FUNCTION_BLOCK FB_SlaveCtrlPrecisionTest EXTENDS FB_SlaveArmCtrlBase
VAR_INPUT
END_VAR
VAR_OUTPUT
END_VAR
VAR
	//arm id
	m_armId:INT;	
	
	//Precision calculation pre matrix
	m_frontPose:ST_Frame;
	
	//Precision calculation post matrix
	m_endPose:ST_Frame;
	
	//single arm pose
	m_slaveArmPose:ST_Frame;
	
	//control mode:  1---Joint space single point motion   2---Continuous joint space motion   3---Single point motion in operating space
	//4---Continuous motion in operating space   5---precision test   6---back to origin position
	m_controlMode:INT:=1;
	
	//test step
	m_testStep:INT;
	
	//DH joint position
	m_initDHPos,m_startDHPos,m_endDHPos :Vec6d;
	
	//startJntPos,endJntPos :Vec8d;
	m_initJntPos,m_startJntPos,m_endJntPos :Vec8d;
	
	//Trajectory planner
	m_Planner: FB_TrajMoveJ;
	
	//motion parameters
	m_maxjntVel,m_maxjntAcc,m_maxjntJerk:Vec8d;
	
	// joint velocity limit
	m_DHJntVel :ARRAY[1..6] OF LREAL :=[1, 1, 0.5, 1,1,1];
	m_maxDHJntVel :ARRAY[1..6] OF LREAL :=[1, 1, 0.5, 1,1,1];	
	m_velFactor:ARRAY[1..2] OF LREAL:=[0.1,1];//lowVel  highVel
	
	//time
	m_time:LREAL;
	
	//joint motion incresement
	m_DHjntInc:Vec6d;
	
	//moiton parameters
	m_jntMotionDir:Vec6i:=[0,0,0,0,0,0];
	m_jntVel:Vec6d:=[0.1,0.1,0.01,0.2,0.2,0.2];
	
	//motion start
	m_startMotion:BOOL;
	m_startMotionLast:BOOL;
	
	//target spatial position
	m_targetSpatialPos:ST_Frame;
	
	//spatial motion parameters
	m_spatialMotionDir:Vec6i;
	m_spatialVel:Vec6d;
	
	//spatial position incresement
	m_spatialPosInc:Vec6d;
	
	//initial spatial position
	m_initSpatialPos:ST_Frame;
	
	//target position variables
	m_posInc:Vec3d;
	m_axis:Vec3d;
	m_angle:LREAL;
	
	//accuracy test variables
	m_pointNum:INT;
	m_pointSum:INT;
	m_motionCycleNum:INT;
	m_targetPosArr:ARRAY[1..5] OF ST_Frame;
	
	//Has the inverse kinematics been successfully solved
	m_IKSucceed:BOOL;	
	
	//Numerical method for inverse solution of related variables
	//m_cmdCartPose:ST_Frame;
	m_slavePosErr :Vec3d;
	m_slaveRotErr :Mat3d;
	m_errAngle : LREAL;
	m_errAxisLocal, m_errAxis :Vec3d;
	m_masterSlavePoseError :Vec6d;
	
	// pose track control kp
	m_posTrackKp :REAL := 100;
	m_oriTrackKp :REAL := 100;
	
	// velocity for slave to track motion
	m_slaveCmdVel, m_slaveCmdWVel : Vec3d;
	invJaco :Mat6d;
	
	//spatial velocity limit
	m_linearVelLimit:LREAL:=0.1;
	m_angularVelLimit:LREAL:=5*g_deg2Rad;
	
	// simulated DH joint position
	m_simDHJntPos : Vec6d;
	
	// simulated slave twist of DH joint
	m_simDHJointVel :Vec6d;
	
	// command joint position filter
	m_cmdJntPosLpf:ARRAY[1..8] OF FB_LowPassFilter;
	
	// filter cut-off frequency for control
	m_macroCmdJntPosLpfCutoffFreq : LREAL :=5;
	m_microCmdJntPosLpfCutoffFreq : LREAL :=15;
	
	//position and posture error limit
	m_distErrLimit:LREAL:=0.001*0.1;
	m_poseErrLimit:LREAL:=0.01*g_deg2Rad;
	m_delayTimeLimit:LREAL:=1;
	m_errTime:LREAL;
	
	//original joint position
	m_originJntPos:Vec6d;
	
	//motion status
	m_motionFinished:BOOL;
END_VAR

METHOD accuracyTest : BOOL
VAR_INPUT
	// slave arm data
	i_slaveArm :FB_SlaveArm;
END_VAR

(*
CASE m_testStep OF
	0: //data initial		
		m_targetSpatialPos:=m_targetPosArr[m_pointNum];
		m_startDHPos:=i_slaveArm.curDHJntPos;
		m_IKSucceed:=i_slaveArm.inverseKinematic(i_targetSpatialPos:= m_targetSpatialPos, i_startDHJntPos:= m_startDHPos, o_outputDHJntPos=> m_endDHPos);
		IF (m_IKSucceed=FALSE) THEN
			m_testStep:=30;
		END_IF
		
		m_startJntPos:=i_slaveArm.curJntPos;	
		i_slaveArm.instrument.instruIK(m_endDHPos,0, o_jntPos=>m_endJntPos);
		m_Planner.init(i_startJntPos:= m_startJntPos, 	i_targetJntPos:= m_endJntPos, 	i_maxJntVel:= m_maxjntVel, 	i_maxJntAcc:= m_maxjntAcc, 	i_maxJntJerk:= m_maxjntJerk);
		IF (m_Planner.isGene=FALSE) THEN
			m_testStep:=30;
		ELSE
			m_time:=0; m_testStep:=10;
		END_IF		
		
		
	10: //start the motion
		m_time:=m_time+g_slaveArmCtrlCycleTime;
		m_Planner.evaluate(t:= m_time, jntPos=> m_cmdJntPos, jntVel=> m_cmdJntVel, jntAcc=> m_cmdJntAcc);
		IF (m_time>m_Planner.duration) THEN
			m_testStep:=20;			
		END_IF
		
		
	20: //Record the motion cycle
		m_pointNum:=m_pointNum+1;
		IF (m_pointNum>m_pointSum) THEN
			m_pointNum:=1;
			m_motionCycleNum:=m_motionCycleNum+1;
			IF (m_motionCycleNum>5) THEN
				m_testStep:=30;
			ELSE
				m_testStep:=0;
			END_IF
		ELSE
			m_testStep:=0;
		END_IF
		
	
	30: //stop
		m_testStep:=-1;		
END_CASE
*)
END_METHOD

METHOD accuracyTest_iter : BOOL
VAR_INPUT
	// slave arm data
	i_slaveArm :FB_SlaveArm;
END_VAR

CASE m_testStep OF
	0: //data initial		
		m_targetSpatialPos:=m_targetPosArr[m_pointNum];
		m_cmdCartPose:=m_targetSpatialPos;
		numericalIK(i_slaveArm);
		
		//Determine if the error is less than the set value
		IF (norm(m_slavePosErr)<m_distErrLimit) AND (m_errAngle<m_poseErrLimit) THEN
			m_errTime:=m_errTime+g_slaveArmCtrlCycleTime;
			IF (m_errTime>m_delayTimeLimit) THEN
				m_errTime:=0;
				m_testStep:=15;
			END_IF
		ELSE
			m_errTime:=0;
		END_IF
	
		
	15: //Waiting for confirmation and measurement
		IF (GVL_AccuracyTestVar.g_nextStep[m_armId]=TRUE) THEN
			GVL_AccuracyTestVar.g_nextStep[m_armId]:=FALSE;
			m_testStep:=20;
		END_IF
		
	
	20: //Record the motion cycle
		m_pointNum:=m_pointNum+1;
		IF (m_pointNum>m_pointSum) THEN
			m_pointNum:=1;
			m_motionCycleNum:=m_motionCycleNum+1;
			IF (m_motionCycleNum>GVL_AccuracyTest.g_testMotCycNum) THEN
				m_testStep:=30;
			ELSE
				m_testStep:=0;
			END_IF
		ELSE
			m_testStep:=0;
		END_IF
	
	
	30: //stop
		m_testStep:=-1;	
		m_motionFinished:=TRUE;	
END_CASE
END_METHOD

METHOD back2origin : BOOL
VAR_INPUT
	// slave arm data
	i_slaveArm :FB_SlaveArm;
END_VAR

CASE m_testStep OF
	0: //Trajectory parameter initialization
		m_startJntPos:=i_slaveArm.curJntPos;
		m_endDHPos:=m_originJntPos;		
		i_slaveArm.instrument.instruIK(m_endDHPos,0, o_jntPos=>m_endJntPos);
		m_Planner.init(i_startJntPos:= m_startJntPos, 	i_targetJntPos:= m_endJntPos, 	i_maxJntVel:= m_maxjntVel, 	i_maxJntAcc:= m_maxjntAcc, 	i_maxJntJerk:= m_maxjntJerk);
		IF (m_Planner.isGene=FALSE) THEN
			m_testStep:=20;
		ELSE
			m_time:=0; m_testStep:=10;
		END_IF		
		
		
	10: //start motion
		m_time:=m_time+g_slaveArmCtrlCycleTime;
		m_Planner.evaluate(t:= m_time, jntPos=> m_cmdJntPos, jntVel=> m_cmdJntVel, jntAcc=> m_cmdJntAcc);
		m_simJntPos:=m_cmdJntPos; //copy value to sim jntpos
		IF (m_time>m_Planner.duration) THEN
			m_testStep:=20;
		END_IF		
		
		
	20: //end the motion
		m_testStep:=-1;		
		m_motionFinished:=TRUE;
END_CASE
END_METHOD

// override this function in each exact controller
METHOD PROTECTED calcCmdJntPos : BOOL
VAR_IN_OUT CONSTANT
	// endoscope pose in cart coordinate
	i_endoscopePose : ST_Frame;
	
	// master arm data
	i_masterStatus :ST_MasterStatus;
	
	// setup arm data
	i_setupStatus: ST_SetupStatus;
	
	// slave arm data
	i_slaveArm :FB_SlaveArm;
END_VAR

VAR
	i:INT;
	tmpFrame:ST_Frame;
	r_angle:LREAL;
END_VAR

//Basic information update---front pose frame and end pose frame 
tmpFrame:=invFrame(i_endoscopePose);
i:=i_slaveArm.armIdx;
m_frontPose:=transform(tmpFrame,i_setupStatus.m_curEndPose[i]);
m_endPose.m_pos:=g_zeroVec3d;  m_endPose.m_rot:=g_eye3d;
m_slaveArmPose:=i_slaveArm.curCartPose;


//copy to global variables
GVL_AccuracyTestVar.g_frontPose[m_armId]:=m_frontPose;
GVL_AccuracyTestVar.g_endPose[m_armId]:=m_endPose;
GVL_AccuracyTestVar.g_slaveArmPose[m_armId]:=m_slaveArmPose;


//Initialization of motion parameters
m_startMotion:=GVL_AccuracyTestVar.g_startMotion[m_armId];
IF (m_startMotionLast=FALSE) AND (m_startMotion=TRUE) THEN
	motionParamInit(i_slaveArm);
END_IF
m_startMotionLast:=m_startMotion;


//Select different programs based on different control modes
IF (m_startMotion=TRUE) THEN
	IF (m_controlMode=1) THEN
		//jntSinglePoint(i_slaveArm);
		
	ELSIF (m_controlMode=2) THEN
		jntContinuousPoint(i_slaveArm);
		
	ELSIF (m_controlMode=3) THEN
		//spaceSinglePoint_iter(i_slaveArm);
		
	ELSIF (m_controlMode=4) THEN
		spaceContinuousPoint_iter(i_slaveArm);
		
	ELSIF (m_controlMode=5) THEN
		accuracyTest_iter(i_slaveArm);
		
	ELSIF (m_controlMode=6) THEN
		back2origin(i_slaveArm);
	END_IF
END_IF


//show the motion step
IF (m_controlMode=5) THEN
	GVL_AccuracyTestVar.g_curStep[m_armId]:=m_testStep;
	GVL_AccuracyTestVar.g_testPointId[m_armId]:=m_pointNum;
	GVL_AccuracyTestVar.g_testCycleId[m_armId]:=m_motionCycleNum;
ELSE
	GVL_AccuracyTestVar.g_curStep[m_armId]:=-1;
	GVL_AccuracyTestVar.g_testPointId[m_armId]:=0;
	GVL_AccuracyTestVar.g_testCycleId[m_armId]:=0;
END_IF



// feedback the motion status
IF (m_controlMode=1) OR (m_controlMode=3) OR (m_controlMode=5) OR (m_controlMode=6) THEN
	IF (m_testStep=-1) AND (m_motionFinished=TRUE) THEN
		m_controlMode:=0;
		GVL_AccuracyTestVar.g_controlMode[m_armId]:=0;	
	END_IF
ELSIF (m_controlMode=2) OR (m_controlMode=4) THEN
	IF (m_startMotion=FALSE) THEN
		m_controlMode:=0;
		GVL_AccuracyTestVar.g_controlMode[m_armId]:=0;
	END_IF
END_IF
END_METHOD

// override this function in each exact controller
// NOTICE: set joint control mode here, and do some initialization if needed
METHOD PUBLIC init : BOOL
VAR_IN_OUT CONSTANT
	i_slaveArm	:FB_SlaveArm;
END_VAR
VAR_IN_OUT 
	r_slaveArmCtrlCmd :ST_SlaveArmCtrlCmds;	
END_VAR

VAR
	
END_VAR
SUPER^.Init(i_slaveArm,r_slaveArmCtrlCmd);

//variable initialization
m_armId:=i_slaveArm.armIdx;

//motion parameters initial
motionParamInit(i_slaveArm);
END_METHOD

METHOD PROTECTED jntContinuousPoint : BOOL
VAR_INPUT
	// slave arm data
	i_slaveArm :FB_SlaveArm;
END_VAR

VAR
	i:INT;
END_VAR

//joint motion incresement calculation
FOR i:=1 TO 6 BY 1 DO
	m_DHjntInc[i]:=m_DHjntInc[i]+m_jntMotionDir[i]*m_jntVel[i]*g_slaveArmCtrlCycleTime;
END_FOR

//determine DH joint position
vecAdd(m_initDHPos,m_DHjntInc,m_endDHPos);
i_slaveArm.instrument.instruIK(m_endDHPos,0, o_jntPos=>m_endJntPos);

//copy the value
m_cmdJntPos:=m_endJntPos;
m_simJntPos:=m_cmdJntPos; //copy value to sim jntpos
END_METHOD

METHOD jntSinglePoint : BOOL
VAR_INPUT
	// slave arm data
	i_slaveArm :FB_SlaveArm;
END_VAR

CASE m_testStep OF
	0: //Trajectory parameter initialization
		m_startJntPos:=i_slaveArm.curJntPos;
		m_endDHPos:=GVL_AccuracyTestVar.g_targetJntPos[m_armId];
		
		i_slaveArm.instrument.instruIK(m_endDHPos,0, o_jntPos=>m_endJntPos);
		m_Planner.init(i_startJntPos:= m_startJntPos, 	i_targetJntPos:= m_endJntPos, 	i_maxJntVel:= m_maxjntVel, 	i_maxJntAcc:= m_maxjntAcc, 	i_maxJntJerk:= m_maxjntJerk);
		IF (m_Planner.isGene=FALSE) THEN
			m_testStep:=20;
		ELSE
			m_time:=0; m_testStep:=10;
		END_IF		
		
		
	10: //start motion
		m_time:=m_time+g_slaveArmCtrlCycleTime;
		m_Planner.evaluate(t:= m_time, jntPos=> m_cmdJntPos, jntVel=> m_cmdJntVel, jntAcc=> m_cmdJntAcc);
		m_simJntPos:=m_cmdJntPos; //copy value to sim jntpos
		IF (m_time>m_Planner.duration) THEN
			m_testStep:=20;
		END_IF		
		
		
	20: //end the motion
		m_testStep:=-1;		
		m_motionFinished:=TRUE;
END_CASE
END_METHOD

METHOD motionParamInit : BOOL
VAR_INPUT
	// slave arm data
	i_slaveArm :FB_SlaveArm;
END_VAR
VAR
	i,j:INT;
	poseVec:Vec6d;
	originPose:ST_Frame;
END_VAR
m_testStep:=0;
m_time:=0;
m_controlMode:=GVL_AccuracyTestVar.g_controlMode[m_armId];
m_motionFinished:=FALSE;


//update the joint velocity
IF (m_controlMode=3) OR (m_controlMode=5) THEN
	vecMultiNum(m_DHJntVel,m_velFactor[1],m_maxDHJntVel); //low velocity
ELSIF (m_controlMode=4) THEN	
	vecMultiNum(m_DHJntVel,m_velFactor[2],m_maxDHJntVel); //high velocity
ELSE
	m_maxDHJntVel:=m_DHJntVel; //original velocity
END_IF


//joint continuous motion parameters
m_initDHPos:=i_slaveArm.curDHJntPos;
m_DHjntInc:=g_zeroVec6d;
m_jntMotionDir:=GVL_AccuracyTestVar.g_jntMotionDir[m_armId];
m_jntVel:=GVL_AccuracyTestVar.g_jntVel[m_armId];
FOR i:=1 TO 6 BY 1 DO
	m_jntVel[i]:=LIMIT(-0.1,m_jntVel[i],0.1);
END_FOR
m_jntVel[3]:=LIMIT(-0.01,m_jntVel[3],0.01);


//spatial continuous motion parameters
m_spatialMotionDir:=GVL_AccuracyTestVar.g_spatialMotionDir[m_armId];
m_spatialVel:=GVL_AccuracyTestVar.g_spatialVel[m_armId];
m_initSpatialPos:=i_slaveArm.curCartPose;
m_spatialPosInc:=g_zeroVec6d;
FOR i:=1 TO 3 BY 1 DO
	m_spatialVel[i]:=LIMIT(-0.01,m_spatialVel[i],0.01);
END_FOR
FOR i:=4 TO 6 BY 1 DO
	m_spatialVel[i]:=LIMIT(-0.1,m_spatialVel[i],0.1);
END_FOR


//velocity---acceleration---jerk
vecMultiNum(GVL_SlaveMotorParameters.g_maxJntVel,0.2,m_maxjntVel);
vecMultiNum(m_maxjntVel,3,m_maxjntAcc);
vecMultiNum(m_maxjntAcc,3,m_maxjntJerk);


//accuracy test variables
m_pointNum:=1;
m_pointSum:=GVL_AccuracyTest.g_testPointNum;
m_motionCycleNum:=1;
m_errTime:=0;


//original joint position
m_originJntPos:=GVL_AccuracyTest.g_originJntPos;


//Obtain the position and posture of the test point location
FOR i:=1 TO 5 BY 1 DO
	FOR j:=1 TO 6 BY 1 DO
		poseVec[j]:=GVL_AccuracyTest.g_testSpacePoint[i,j];
	END_FOR
	xyzrpy2Frame(i_posVec:= poseVec, o_frame=> m_targetPosArr[i]);
	
	i_slaveArm.forwardKinematic(i_DHJntPos:= m_originJntPos, r_cartPose:= originPose);
	m_targetPosArr[i].m_rot:=originPose.m_rot;
END_FOR


// init filter
FOR i:=1 TO 3 DO
	m_cmdJntPosLpf[i].init(1, m_macroCmdJntPosLpfCutoffFreq, g_slaveArmCtrlFreq);
END_FOR
FOR i:=4 TO g_sJntNum DO
	m_cmdJntPosLpf[i].init(1, m_microCmdJntPosLpfCutoffFreq, g_slaveArmCtrlFreq);
END_FOR
END_METHOD

METHOD numericalIK : BOOL
VAR_INPUT
	// slave arm data
	i_slaveArm :FB_SlaveArm;
END_VAR

VAR
	i:INT;
	tmpMat3d:Mat3d;
	linearVelScale:LREAL;
	angularVelScale:LREAL;
END_VAR

		//Solve the error term
		vecSub(m_cmdCartPose.m_pos, i_slaveArm.simCartPose.m_pos, m_slavePosErr);
		matTranspose(i_slaveArm.simCartPose.m_rot, tmpMat3d);
		matMultiply(tmpMat3d, m_cmdCartPose.m_rot, m_slaveRotErr);
		rot2AngAxis(m_slaveRotErr, angle=>m_errAngle, axis=>m_errAxisLocal);
		matMultiVec(i_slaveArm.simCartPose.m_rot, m_errAxisLocal, m_errAxis);
		
		// pose track control
		vecMultiNum(m_slavePosErr, m_posTrackKp, m_slaveCmdVel);
		vecMultiNum(m_errAxis, m_errAngle*m_oriTrackKp, m_slaveCmdWVel);
		
		
		//Limit spatial linear velocity and angular velocity
		linearVelScale:=norm(m_slaveCmdVel)/m_linearVelLimit;
		angularVelScale:=norm(m_slaveCmdWVel)/m_angularVelLimit;	
		IF (linearVelScale)>1 THEN
			vecSelfMultiNum(m_slaveCmdVel,1.0/linearVelScale);
		END_IF
		IF (angularVelScale)>1 THEN
			vecSelfMultiNum(m_slaveCmdWVel,1.0/angularVelScale);
		END_IF
		
		
		// final command twist
		FOR i:=1 TO 3 DO 
			m_cmdCartTwist[i] := m_slaveCmdVel[i];
			m_cmdCartTwist[i+3] := m_slaveCmdWVel[i];
		END_FOR
		
		// compute command velocity for DH joints
		invJaco := i_slaveArm.simJacoInv;
		matMultiVec(invJaco, m_cmdCartTwist, m_simDHJointVel);
		
		// limit DH joints velocity and integrate command DH joint position
		FOR i:=1 TO 6 DO 
			m_simDHJointVel[i] := LIMIT(-m_maxDHJntVel[i], m_simDHJointVel[i], m_maxDHJntVel[i]);
			
			m_simDHJntPos[i] := i_slaveArm.simDHJntPos[i] + m_simDHJointVel[i]*g_slaveArmCtrlCycleTime;
			IF (m_simDHJntPos[i]>GVL_SlaveMotorParameters.g_maxDHJntPos[i]) OR (m_simDHJntPos[i]<GVL_SlaveMotorParameters.g_minDHJntPos[i]) THEN
				m_simDHJointVel[i]:=0;
				m_simDHJntPos[i] := i_slaveArm.simDHJntPos[i];
			END_IF
		END_FOR
		
		// calculate target motor joint position/velocity from DH joint position
		i_slaveArm.instrument.instruIK(m_simDHJntPos,0, o_jntPos=>m_simJntPos);
		
		// filt command joint position
		FOR i:=1 TO g_sJntNum DO 
			//m_cmdJntPos[i] := m_cmdJntPosLpf[i].run(m_simJntPos[i]);
		END_FOR
		m_cmdJntPos:=m_simJntPos;
END_METHOD

METHOD rpy2rot : BOOL
VAR_INPUT
	i_rpy:Vec3d;
END_VAR

VAR_OUTPUT
	o_rot:Mat3d;
END_VAR

VAR
	rot_x,rot_y,rot_z:LREAL;
	alpha,beta,gama:LREAL;
	matrix_out:ARRAY[1..3,1..3] OF LREAL;
END_VAR

alpha:=rot_z;
beta:=rot_y;
gama:=rot_x;

matrix_out[1,1]:=COS(alpha)*COS(beta);
matrix_out[2,1]:=SIN(alpha)*COS(beta);
matrix_out[3,1]:=-SIN(beta);

matrix_out[1,2]:=COS(alpha)*SIN(beta)*SIN(gama)-SIN(alpha)*COS(gama);
matrix_out[2,2]:=SIN(alpha)*SIN(beta)*SIN(gama)+COS(alpha)*COS(gama);
matrix_out[3,2]:=COS(beta)*SIN(gama);

matrix_out[1,3]:=COS(alpha)*SIN(beta)*COS(gama)+SIN(alpha)*SIN(gama);
matrix_out[2,3]:=SIN(alpha)*SIN(beta)*COS(gama)-COS(alpha)*SIN(gama);
matrix_out[3,3]:=COS(beta)*COS(gama);

o_rot:=matrix_out;
END_METHOD

METHOD spaceContinuousPoint : BOOL
VAR_INPUT
	// slave arm data
	i_slaveArm :FB_SlaveArm;
END_VAR

VAR
	i:INT;	
	rotMatrix:Mat3d;
	tmpFrame:ST_Frame;
END_VAR
(*
//spatial motion incresement calculation
FOR i:=1 TO 6 BY 1 DO
	m_spatialPosInc[i]:=m_spatialPosInc[i]+m_spatialMotionDir[i]*m_spatialVel[i]*g_slaveArmCtrlCycleTime;
END_FOR


//Calculate the target pose matrix
FOR i:=1 TO 3 BY 1 DO
	m_posInc[i]:=m_spatialPosInc[i];
	m_axis[i]:=m_spatialVel[i];
END_FOR
m_angle:=norm(m_spatialPosInc);
tmpFrame.m_pos:=m_posInc;
tmpFrame.m_rot:=angAxis2Rot(m_angle,m_axis);
m_targetSpatialPos:=transform(m_initSpatialPos,tmpFrame);

//Inverse kinematics solution of surgical arm
m_startDHPos:=i_slaveArm.curDHJntPos;
m_IKSucceed:=i_slaveArm.inverseKinematic(i_targetSpatialPos:= tmpFrame, i_startDHJntPos:= m_startDHPos, o_outputDHJntPos=> m_endDHPos);
IF (m_IKSucceed=FALSE) THEN
	RETURN;
END_IF

//determine joint position
i_slaveArm.instrument.instruIK(m_endDHPos,0, o_jntPos=>m_endJntPos);
m_cmdJntPos:=m_endJntPos;
*)
END_METHOD

METHOD spaceContinuousPoint_iter : BOOL
VAR_INPUT
	// slave arm data
	i_slaveArm :FB_SlaveArm;
END_VAR

VAR
	i:INT;	
	rotMatrix:Mat3d;
	tmpFrame:ST_Frame;
	testVec6d:Vec6d;
END_VAR

//spatial motion incresement calculation
FOR i:=1 TO 6 BY 1 DO
	m_spatialPosInc[i]:=m_spatialPosInc[i]+m_spatialMotionDir[i]*m_spatialVel[i]*g_slaveArmCtrlCycleTime;
END_FOR

//Calculate the target pose matrix
FOR i:=1 TO 3 BY 1 DO
	m_posInc[i]:=m_spatialPosInc[i];
	m_axis[i]:=m_spatialMotionDir[i+3];
END_FOR
m_angle:=norm(m_spatialPosInc);
tmpFrame.m_pos:=m_posInc;
tmpFrame.m_rot:=angAxis2Rot(m_angle,m_axis);
m_targetSpatialPos:=transform(m_initSpatialPos,tmpFrame);

// Numerical method for inverse solution
m_cmdCartPose:=m_targetSpatialPos;
numericalIK(i_slaveArm);
END_METHOD

METHOD spaceSinglePoint : BOOL
VAR_INPUT
	// slave arm data
	i_slaveArm :FB_SlaveArm;
END_VAR

(*
CASE m_testStep OF
	0: //Trajectory parameter initialization
		m_targetSpatialPos:=GVL_AccuracyTestVar.g_targetSpatialPos[m_armId];
		m_startDHPos:=i_slaveArm.curDHJntPos;
		m_IKSucceed:=i_slaveArm.inverseKinematic(i_targetSpatialPos:= m_targetSpatialPos, i_startDHJntPos:= m_startDHPos, o_outputDHJntPos=> m_endDHPos);
		IF (m_IKSucceed=FALSE) THEN
			m_testStep:=20;
		END_IF
		
		m_startJntPos:=i_slaveArm.curJntPos;		
		i_slaveArm.instrument.instruIK(m_endDHPos,0, o_jntPos=>m_endJntPos);
		m_Planner.init(i_startJntPos:= m_startJntPos, 	i_targetJntPos:= m_endJntPos, 	i_maxJntVel:= m_maxjntVel, 	i_maxJntAcc:= m_maxjntAcc, 	i_maxJntJerk:= m_maxjntJerk);
		IF (m_Planner.isGene=FALSE) THEN
			m_testStep:=20;
		ELSE
			m_time:=0; m_testStep:=10;
		END_IF		
		
		
	10: //start motion
		m_time:=m_time+g_slaveArmCtrlCycleTime;
		m_Planner.evaluate(t:= m_time, jntPos=> m_cmdJntPos, jntVel=> m_cmdJntVel, jntAcc=> m_cmdJntAcc);
		IF (m_time>m_Planner.duration) THEN
			m_testStep:=20;
		END_IF		
		
		
	20: //end the motion
		m_testStep:=-1;		
END_CASE
*)
END_METHOD

METHOD spaceSinglePoint_iter : BOOL
VAR_INPUT
	// slave arm data
	i_slaveArm :FB_SlaveArm;
END_VAR

VAR
	tmpMat3d:Mat3d;
	i:INT;
END_VAR

CASE m_testStep OF
	0: //Numerical method for inverse solution
		m_targetSpatialPos:=GVL_AccuracyTestVar.g_targetSpatialPos[m_armId];
		m_cmdCartPose:=m_targetSpatialPos;
		numericalIK(i_slaveArm);
		
		//Determine if the error is less than the set value
		IF (norm(m_slavePosErr)<m_distErrLimit) AND (m_errAngle<m_poseErrLimit) THEN
			m_errTime:=m_errTime+g_slaveArmCtrlCycleTime;
			IF (m_errTime>m_delayTimeLimit) THEN
				m_errTime:=0;
				m_testStep:=10;
			END_IF
		ELSE
			m_errTime:=0;
		END_IF
		
		
	10: //end the motion
		m_testStep:=-1;	
		m_motionFinished:=TRUE;	
END_CASE
END_METHOD

METHOD xyzrpy2Frame : BOOL
VAR_INPUT
	i_posVec:Vec6d;
END_VAR

VAR_OUTPUT
	o_frame:ST_Frame;
END_VAR

VAR
	i:INT;
	rpyVec:Vec3d;
END_VAR

FOR i:=1 TO 3 BY 1 DO
	o_frame.m_pos[i]:=i_posVec[i];
	rpyVec[i]:=i_posVec[i+3];
END_FOR
rpy2rot(i_rpy:= rpyVec, o_rot=> o_frame.m_rot) ;
END_METHOD

END_FUNCTION_BLOCK

(* stored: Version 1.1.0.1, ProductVersion 3.1.4024.11
   POU FB_SlaveCtrlPrecisionTest: Id {1902434d-be0a-47a5-87d4-f277642374f0}, SpecialFunc None
   Method accuracyTest: Id {3de375b6-4f4e-4ec7-8c4b-4769583261f7}
   Method accuracyTest_iter: Id {0a89f2b7-69f4-48e8-9e4f-4df31d757009}
   Method back2origin: Id {9ec190e9-bfb3-4e1c-bdd7-56aa92acda9b}
   Method calcCmdJntPos: Id {45ff5261-3263-4c0a-bada-e4386f88b1cb}
   Method init: Id {0d0573e4-bcf6-41e5-aaae-f56a6c51570f}
   Method jntContinuousPoint: Id {fbcb4435-cae6-4265-9904-f0248e46b86e}
   Method jntSinglePoint: Id {0dd167e7-64df-41a9-986a-68e28cb0e649}
   Method motionParamInit: Id {307213d8-b11a-481a-bd29-12db6287c686}
   Method numericalIK: Id {338e4e28-3e43-4c80-8233-1764e66a46e4}
   Method rpy2rot: Id {2a77c0e7-fd72-47f1-a5e9-51bdfe702e1b}
   Method spaceContinuousPoint: Id {3ae3ce74-e097-4489-b011-9dcbcf97ed0f}
   Method spaceContinuousPoint_iter: Id {a761fe40-0c83-4c79-9e02-31b1555561ae}
   Method spaceSinglePoint: Id {57935730-d3e0-49a0-a5e7-5322f40a77c8}
   Method spaceSinglePoint_iter: Id {e95481d5-fc1a-4f39-b6aa-ed5875ff2314}
   Method xyzrpy2Frame: Id {386a3d45-d2c1-4c32-a59e-a596651a6100} *)
